// TIA Portal V20 export
FUNCTION_BLOCK "CC_Pneumatic_Roller"   // FB104, LAD
{ S7_Optimized_Access := 'TRUE' }
// stored: AutoNumber false, MemoryReserve 100, SetENOAutomatically false
   VAR_INPUT
      ReqUp : Bool;
      ReqDown : Bool;
      Sensor1Down : Bool;
      Sensor1Up : Bool;
      Sensor2Down : Bool;
      Sensor2Up : Bool;
      Interlock : Bool;
      Timeout : Time := T#3s;
   END_VAR
   VAR_OUTPUT
      Valve : Bool;
      Error : Bool;
      "Step" : Int;
      PosUp : Bool;
      PosDown : Bool;
   END_VAR
   VAR
      IEC_Timout_retracting { S7_SetPoint := 'True'} : TOF_TIME;
      IEC_Timout_extracting { S7_SetPoint := 'True'} : TON_TIME;
   END_VAR
   VAR CONSTANT
      STEP_RETRACT : Int := 1;
      STEP_MOVING : Int := 2;
      STEP_EXTEND : Int := 3;
   END_VAR
BEGIN

REGION Network 1
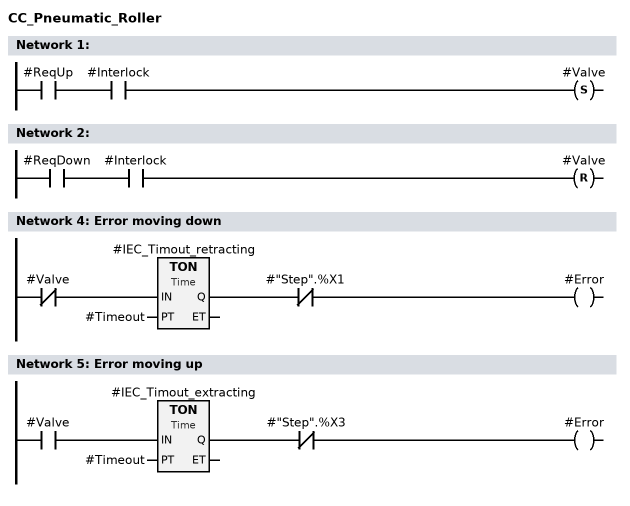
   RUNG wire#powerrail
      Contact( #ReqUp )
      Contact( #Interlock )
      S_Coil( #Valve )
   END_RUNG
   // the same network as SCL:
   IF #ReqUp AND #Interlock THEN #Valve := TRUE; END_IF;
END_REGION

REGION Network 2
   RUNG wire#powerrail
      Contact( #ReqDown )
      Contact( #Interlock )
      R_Coil( #Valve )
   END_RUNG
   // the same network as SCL:
   IF #ReqDown AND #Interlock THEN #Valve := FALSE; END_IF;
END_REGION

REGION Network 3 (SCL)
   #PosDown := FALSE;
   #PosUp := FALSE;
   #Step := 0;
   IF #Sensor1Down = 0 AND #Sensor1Up = 1 AND #Sensor2Down = 0 AND #Sensor2Up = 1 THEN
       #Step.%X3 :=1;
       #PosUp := True;
   ELSIF #Sensor1Down AND #Sensor1Up = 0 AND #Sensor2Down AND #Sensor2Up = 0 THEN
       #Step.%X1 := 1;
       #PosDown := True;
   ELSE
       #Step.%X2:= 1;
   END_IF;
END_REGION

REGION Network 4: Error moving down
   RUNG wire#powerrail
      I_Contact( #Valve )
      { S7_Templates := "time_type := Time" } #IEC_Timout_retracting.TON(pt := #Timeout, et =>)
      I_Contact( #"Step".%X1 )
      Coil( #Error )
   END_RUNG
   // the same network as SCL:
   #IEC_Timout_retracting(IN := NOT #Valve, PT := #Timeout);   // TON
   #Error := #IEC_Timout_retracting.Q AND NOT #"Step".%X1;
END_REGION

REGION Network 5: Error moving up
   RUNG wire#powerrail
      Contact( #Valve )
      { S7_Templates := "time_type := Time" } #IEC_Timout_extracting.TON(pt := #Timeout, et =>)
      I_Contact( #"Step".%X3 )
      Coil( #Error )
   END_RUNG
   // the same network as SCL:
   #IEC_Timout_extracting(IN := #Valve, PT := #Timeout);   // TON
   #Error := #IEC_Timout_extracting.Q AND NOT #"Step".%X3;
END_REGION
END_FUNCTION_BLOCK
